# EPICS alarm handler configuration: mps_database/bareTest/alarms/areas/mpln_undh_mp03.alhConfig
GROUP NULL MPLN:UNDH:MP03:1
$ALIAS MPS Link Node 138
$GUIDANCE
LTUH MPS
   Group Name: MPLN:UNDH:MP03:1
   Summary PV:  MPLN:UNDH:MP03:1:STATSUMY
$END
CHANNEL  MPLN:UNDH:MP03:1    MPLN:UNDH:MP03:1:MPS_EN_RBV		-----
CHANNEL  MPLN:UNDH:MP03:1    MPLN:UNDH:MP03:1:LC1_MODE_RBV		-----
